// TIA Portal V16 export
// export: Created 2024-12-03T15:41:43.112528Z, ExportSetting WithDefaults, DisplayName Totally Integrated Automation Portal, DisplayVersion V16 Update 6, DisplayName TIA Portal Version Control Interface, DisplayVersion V16 Update 2, DisplayName TIA Portal Openness, DisplayVersion V16 Update 6, DisplayName TIA Portal Teamcenter Gateway, DisplayVersion V16, DisplayName SINAMICS Startdrive Advanced, DisplayVersion V16 Update 5, DisplayName SINAMICS Startdrive G130, G150, S120, S150, SINAMICS MV, S210, DisplayVersion V16 Update 5, DisplayName SINAMICS Startdrive G110M, G120, G120C, G120D, G120P, G115D, DisplayVersion V16 Update 5, DisplayName STEP 7 Professional, DisplayVersion V16 Update 6, DisplayName STEP 7 Safety, DisplayVersion V16, DisplayName WinCC Advanced / Unified PC, DisplayVersion V16 Update 6
FUNCTION_BLOCK "Gravity_Conveyor_Controller_FB"   // FB68, SCL
{ S7_Optimized_Access := 'TRUE' }
VERSION : 0.1
// stored: AutoNumber true, IsIECCheckEnabled false, IsRetainMemResEnabled false, MemoryReserve 100, SetENOAutomatically false, UDAEnableTagReadback false
   VAR_INPUT
      I_BuildName : Bool := true;
      I_Upstream : "Conveyor_UDT";
      I_ConnectUpstream : Bool;
      I_PC : "IPC_ROUTING_DATA_UDT";
   END_VAR
   VAR_IN_OUT
      IO_Conv : "Conveyor_UDT";
      IO_IPC : "PLC_ROUTING_DATA_UDT";
   END_VAR
   VAR
      ipc : "IPC_Request";
      cyclerun : "CycleRun";
      fullDetection { S7_SetPoint := 'True'} : TON_TIME;
      Alarm : "AlarmInfo_UDT";
      AlarmInfoValue : String;
      BlockAlarm { S7_SetPoint := 'True'} : Program_Alarm;
   END_VAR
   VAR_TEMP
      T_Data : "PLC_GETDATA_REQ_DATA_UDT";
      T_ZoneInfo : "ZoneInfo";
      T_Appstate : "ApplicationState_UDT";
      T_Condition : Bool;
   END_VAR
BEGIN
   #T_ZoneInfo := "ApplicationState_DB".ZoneNames[#IO_Conv.Zone];
   #T_Appstate := "ApplicationState_DB".Appstate[#T_ZoneInfo.AppStateIndex];
   #IO_Conv.Status.StartedAutoMode := #T_Appstate.States.AutoModeActivated.State;
   #cyclerun();

   #IO_Conv.Settings.Timings.ReceiveDistance := 3;

   REGION Empty

       #IO_Conv.Status.Empty := NOT #IO_Conv.Input.SensorAtEndLogic.State;

   END_REGION

   REGION TRACKING

       #IO_Conv.Status.ObjectReceivePulse := 0;

       IF #I_Upstream.Status.ObjectSentPulse AND #I_ConnectUpstream AND
           #I_Upstream.Input.Running_FB THEN
           #IO_Conv.TrackingStat.Current := #I_Upstream.TrackingStat.InSending;
           #IO_Conv.TrackingStat.Current.Barcode := #I_Upstream.TrackingStat.InSending.Barcode;
           #IO_Conv.Status.ObjectReceivePulse := 1;
       END_IF;

   END_REGION

   REGION IPC

       #T_Data.barcode := #IO_Conv.TrackingStat.Current.Barcode;
       #T_Data.weightGrams := 0;

       #ipc(I_StartRequestFlag:=#IO_Conv.Status.ObjectReceivePulse,
            I_Data:=#T_Data,
            I_ResStatus:=#I_PC.RES_STATUS,
            I_ResData:=#I_PC.RES_DATA,
            IO_IPC_Interface:=#IO_IPC.IPC_STATUS,
            IO_ReqStatus:=#IO_IPC.REQ_STATUS,
            IO_ReqData:=#IO_IPC.REQ_DATA,
            IO_ResultData:=#IO_IPC.PLC_DATA);

   END_REGION

   REGION Ready TO receive

       IF NOT #IO_Conv.Input.SensorAtEndLogic.State THEN
           #IO_Conv.Cmd.ReadyToReceive := true;
       END_IF;


       IF #fullDetection.Q AND NOT #I_Upstream.Cmd.RunAuto THEN
           #IO_Conv.Cmd.ReadyToReceive := FALSE;
       END_IF;


   END_REGION

   REGION Ready TO sent

       #IO_Conv.Cmd.ReadyToSent := #IO_Conv.Input.SensorAtEndLogic.State;

   END_REGION

   REGION Always run

       #IO_Conv.Cmd.RunAuto := #IO_Conv.Cmd.ReadyToReceive;
       #IO_Conv.Input.Running_FB := #IO_Conv.Cmd.RunAuto;

   END_REGION

   REGION alarms

       REGION CONV NAME

           IF NOT #Alarm.init AND #I_BuildName THEN
               #IO_Conv.Name := "buildObjectName"(I_Symbolname := GetSymbolName(variable := #IO_Conv, size := 100));
               #Alarm.info := "buildAlarmInfo"(I_ObjectName := #IO_Conv.Name, I_ZoneIndex := #IO_Conv.Zone, I_ZoneName := #T_ZoneInfo.ZoneName);
               #Alarm.init := true;
           END_IF;

       END_REGION

       REGION CONVEYOR FULL

           #IO_Conv.Settings.Timings.ReceiveDistance := 4;
           #IO_Conv.Settings.Alarms.BlockDetectionOn := 1;

           #T_Condition :=
           #IO_Conv.Input.SensorAtEndLogic.State AND
           #IO_Conv.Settings.Alarms.BlockDetectionOn
           AND #T_Appstate.States.AutoModeActivated.State AND
           NOT "Simulation_DB".ByPassGravityConv;


           #fullDetection(IN := #T_Condition,
                          PT := REAL_TO_DINT(#IO_Conv.Settings.Timings.ReceiveDistance * 1000));
       END_REGION

       #IO_Conv.Alarms.Status.%X0 :=
       #IO_Conv.Alarms.BlockedReceive.Active := #fullDetection.Q;

       REGION ALARM ACTIVE

           #IO_Conv.Alarms.AlarmActive.Active := #IO_Conv.Alarms.Status > 0;

           // IF #IO_Conv.Alarms.Status > 0 THEN
           //     "ApplicationState_DB".Appstate[#T_ZoneInfo.AppStateIndex].Alarms.AlarmActiveInternalPLC := TRUE;
           // END_IF;

       END_REGION

       REGION PROGRAM ALARM
           IF #cyclerun.O_Cycle = 10 THEN
               #BlockAlarm(SIG := #fullDetection.Q AND false,
                           SD_1 := #Alarm.info,
                           SD_2 := #T_ZoneInfo.ZoneName,
                           SD_3 := #IO_Conv.Name);
           END_IF;
       END_REGION

   END_REGION
END_FUNCTION_BLOCK
